(* PLC project CoDeSys External Library Template, WAGO e!COCKPIT e!COCKPIT, author 3S - Smart Software Solutions GmbH *)
(* stored: creationDateTime 2019-10-29T12:37:19.7399039, version 3.5.5.30, modificationDateTime 2019-10-29T12:36:39.3744516, organization 3S - Smart Software Solutions GmbH *)
(* Library project template with all possible element types, docu and a sample project structure *)

FUNCTION_BLOCK fbTimer
  VAR_INPUT
    xWejscie : BOOL;
    tCzas : TIME;
    tCzasOn : TIME;
    tCzasOff : TIME;
    xReset : BOOL;
    intTyp : INT;
  END_VAR
  VAR_OUTPUT
    xWyjscie : BOOL;
    xError : BOOL;
  END_VAR
  VAR
    negZboczeOpadajace : F_TRIG;
    tCzasowka1 : TON;
    tCzasowka2 : TON;
    xCzasowka1Wyzwolona : BOOL;
    xCzasowka2Wyzwolona : BOOL;
    xCzasowkaStartup : BOOL := TRUE;
  END_VAR

            // Funkcja rozszerzająca funkcjonalność timera

// intTyp - 1 - Opóźnienie włączenia

// xWejscie - sygnał wejściowy zostanie opóźniony na wyjściu xWyjscie po czasie tCzas
// xReset - resetuje czasówkę wznowienie liczenia czasu po powrocie xReset do FALSE
// tCzas - Czas opóźnienia
// tCzasOn - Czas aktywnego wyjścia T#0s - nieskończoność

// intTyp = 2 - Pulse generator

// xWejscie - aktywuje działanie bloku
// tCzasOn - ile czasu xWyjscie ma byc TRUE - jeśli czas = T#0s stan TRUE pojawia się na jeden skan programu
// tCzasOff - ile czasu xWyjscie ma byc FALSE - jeśli czas = T#0s stan FALSE pojawia się na jeden skan programu

// intTyp = 3 - Pulse
// xWejscie - po pojawieniu się xWejscie przez czas tCzas XWyjscie będzie aktywne

// intTyp = 4 -delayed off
// xWejscie aktywne - xWyjscie aktywne, xWejscie deaktywacja - xWyjscie deaktywacja po tCzas

CASE intTyp OF

	1: 
	tCzasowka1(IN:=xWejscie AND NOT xReset,PT:=tCzas);
	IF tCzasOn = T#0S THEN
		xWyjscie := tCzasowka1.Q;
		ELSE
		tCzasowka2(IN := tCzasowka1.Q , PT := tCzasOn);
		xWyjscie := tCzasowka1.Q AND NOT tCzasowka2.Q;
	END_IF

	2:
	tCzasowka1(IN :=  xWejscie AND NOT tCzasowka2.Q , PT := tCzasOff);
	tCzasowka2(IN :=  xWejscie AND tCzasowka1.Q , PT := tCzasOn);
	xWyjscie := tCzasowka1.Q;
		
	3:
	negZboczeOpadajace(CLK := xWejscie);
	tCzasowka1(IN:= xWejscie OR negZboczeOpadajace.Q , PT := tCzas);
	xWyjscie := (xWejscie OR negZboczeOpadajace.Q) AND NOT tCzasowka1.Q;
	
	4:
	negZboczeOpadajace(CLK := xWejscie);
	IF negZboczeOpadajace.Q THEN
		xCzasowkaStartup := FALSE;
	END_IF
	tCzasowka1(IN := NOT negZboczeOpadajace.Q , PT := tCzas);
	xWyjscie := xWejscie OR (NOT tCzasowka1.Q AND NOT xCzasowkaStartup);
	ELSE
		xError := TRUE;
END_CASE;
          
END_FUNCTION_BLOCK
